// Mitsubishi GX Developer project: fx2cn   PLC: FX2N

PROGRAM MAIN
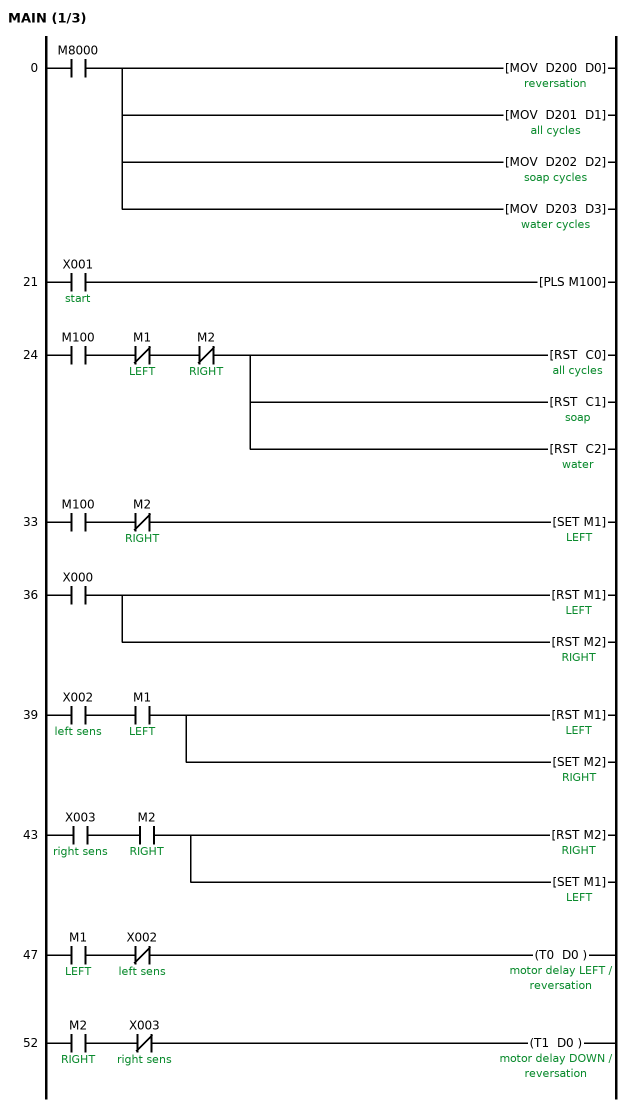
0     LD      M8000
      MOV     D200 D0  ; reversation
      MOV     D201 D1  ; all cycles
      MOV     D202 D2  ; soap cycles
      MOV     D203 D3  ; water cycles
21    LD      X001  ; start
      PLS     M100
24    LD      M100
      ANI     M1  ; LEFT
      ANI     M2  ; RIGHT
      RST     C0  ; all cycles
      RST     C1  ; soap
      RST     C2  ; water
33    LD      M100
      ANI     M2  ; RIGHT
      SET     M1  ; LEFT
36    LD      X000
      RST     M1  ; LEFT
      RST     M2  ; RIGHT
39    LD      X002  ; left sens
      AND     M1  ; LEFT
      RST     M1  ; LEFT
      SET     M2  ; RIGHT
43    LD      X003  ; right sens
      AND     M2  ; RIGHT
      RST     M2  ; RIGHT
      SET     M1  ; LEFT
47    LD      M1  ; LEFT
      ANI     X002  ; left sens
      OUT     T0 D0  ; motor delay LEFT / reversation
52    LD      M2  ; RIGHT
      ANI     X003  ; right sens
      OUT     T1 D0  ; motor delay DOWN / reversation
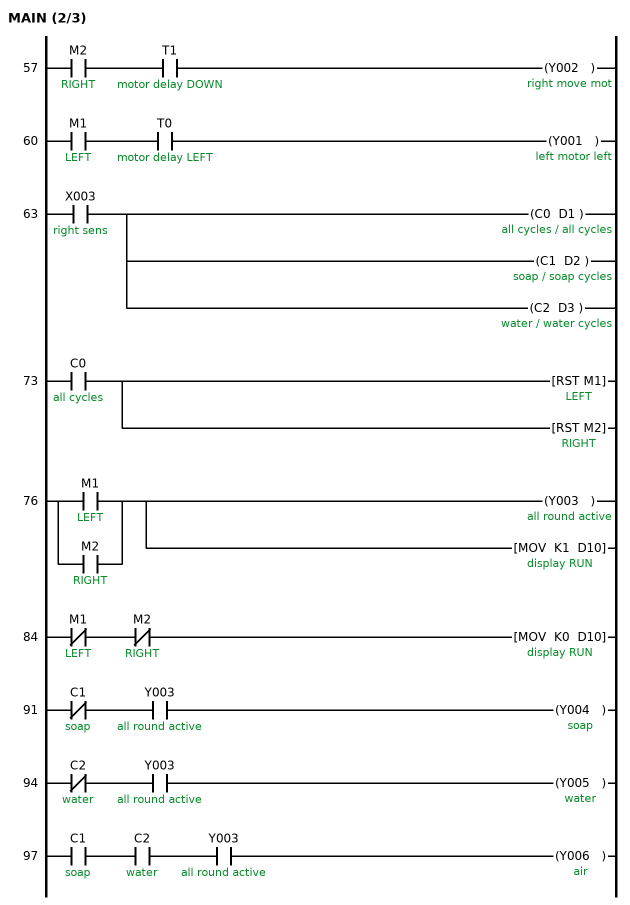
57    LD      M2  ; RIGHT
      AND     T1  ; motor delay DOWN
      OUT     Y002  ; right move mot
60    LD      M1  ; LEFT
      AND     T0  ; motor delay LEFT
      OUT     Y001  ; left motor left
63    LD      X003  ; right sens
      OUT     C0 D1  ; all cycles / all cycles
      OUT     C1 D2  ; soap / soap cycles
      OUT     C2 D3  ; water / water cycles
73    LD      C0  ; all cycles
      RST     M1  ; LEFT
      RST     M2  ; RIGHT
76    LD      M1  ; LEFT
      OR      M2  ; RIGHT
      OUT     Y003  ; all round active
      MOV     K1 D10  ; display RUN
84    LDI     M1  ; LEFT
      ANI     M2  ; RIGHT
      MOV     K0 D10
91    LDI     C1  ; soap
      AND     Y003  ; all round active
      OUT     Y004  ; soap
94    LDI     C2  ; water
      AND     Y003  ; all round active
      OUT     Y005  ; water
97    LD      C1  ; soap
      AND     C2  ; water
      AND     Y003  ; all round active
      OUT     Y006  ; air
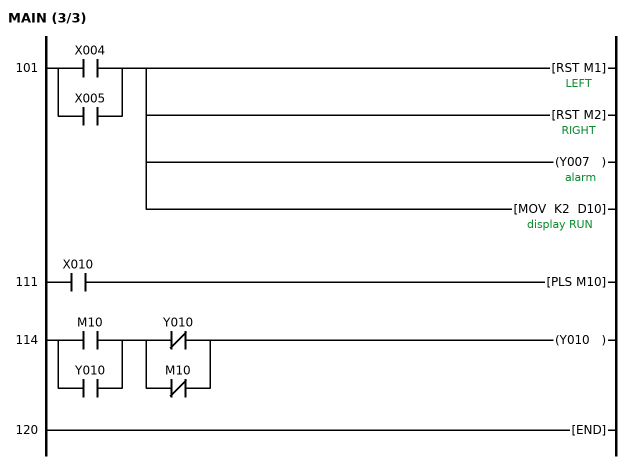
101   LD      X004
      OR      X005
      RST     M1  ; LEFT
      RST     M2  ; RIGHT
      OUT     Y007  ; alarm
      MOV     K2 D10
111   LD      X010
      PLS     M10
114   LD      M10
      OR      Y010
      LDI     Y010
      ORI     M10
      ANB
      OUT     Y010
120   END
END_PROGRAM
